TYPE ST_LoadingStation_InOuts :
STRUCT
	bBottleDetectedSensor AT %I*:BOOL;
	bConveyorIsWorking AT %I*:BOOL;
	rConveyorSpeedControl AT %Q*:REAL;
	
END_STRUCT
END_TYPE

(* stored: Version 1.1.0.1, ProductVersion 3.1.4024.15
   DUT ST_LoadingStation_InOuts: Id {675a0f29-2949-4371-bd1a-150550b89c80} *)
